TYPE T_OCV_Filename : T_MaxString;
END_TYPE

(* stored: Version 1.1.0.1
   DUT T_OCV_Filename: Id {d2e1d0ef-d3d8-44e6-9985-d105c23d3f2a} *)
